// Mitsubishi GX Works2 project: TIMEREX2   PLC: Q03UDV

PROGRAM MAIN
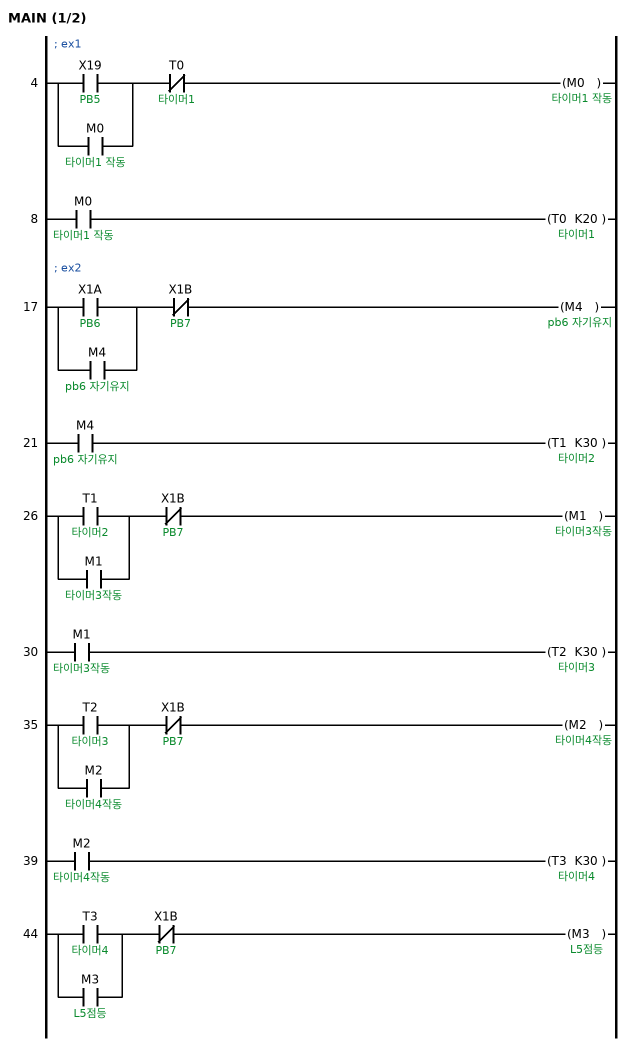
; ex1
4     LD      X19  ; PB5
      OR      M0  ; 타이머1 작동
      ANI     T0  ; 타이머1
      OUT     M0  ; 타이머1 작동
8     LD      M0  ; 타이머1 작동
      OUT     T0 K20  ; 타이머1
; ex2
17    LD      X1A  ; PB6
      OR      M4  ; pb6 자기유지
      ANI     X1B  ; PB7
      OUT     M4  ; pb6 자기유지
21    LD      M4  ; pb6 자기유지
      OUT     T1 K30  ; 타이머2
26    LD      T1  ; 타이머2
      OR      M1  ; 타이머3작동
      ANI     X1B  ; PB7
      OUT     M1  ; 타이머3작동
30    LD      M1  ; 타이머3작동
      OUT     T2 K30  ; 타이머3
35    LD      T2  ; 타이머3
      OR      M2  ; 타이머4작동
      ANI     X1B  ; PB7
      OUT     M2  ; 타이머4작동
39    LD      M2  ; 타이머4작동
      OUT     T3 K30  ; 타이머4
44    LD      T3  ; 타이머4
      OR      M3  ; L5점등
      ANI     X1B  ; PB7
      OUT     M3  ; L5점등
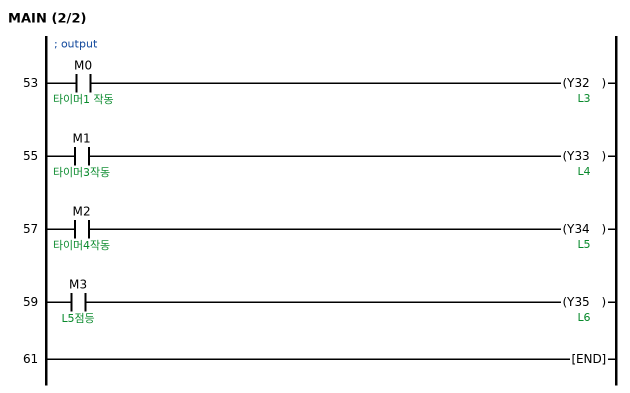
; output
53    LD      M0  ; 타이머1 작동
      OUT     Y32  ; L3
55    LD      M1  ; 타이머3작동
      OUT     Y33  ; L4
57    LD      M2  ; 타이머4작동
      OUT     Y34  ; L5
59    LD      M3  ; L5점등
      OUT     Y35  ; L6
61    END
END_PROGRAM
